FUNCTION_BLOCK SPLIT_AW_INTO_AB (* this Function splits the 2 AB (BYTE) adapters from a AW (WORD) *)
  (* Standard: 61499-2; Description: Copyright (c) 2026 Meisterschulen am Ostbahnhof SPDX-License-Identifier: EPL-2.0 *)
  (* Version 1.0, 2026-05-16, Franz Höpfinger, Meisterschulen am Ostbahnhof, initial API and implementation and/or initial documentation *)
  PACKAGE adapter::splitting;
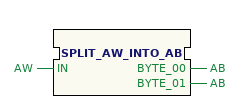
  SOCKETS
    IN : adapter::types::unidirectional::AW; (* WORD Input *)
  END_SOCKETS
  PLUGS
    BYTE_00 : adapter::types::unidirectional::AB; (* Byte 0 *)
    BYTE_01 : adapter::types::unidirectional::AB; (* Byte 1 *)
  END_PLUGS
END_FUNCTION_BLOCK
